INTERFACE I_DigitalInput EXTENDS I_Channel

PROPERTY P_Value : bool
GET
END_GET
END_PROPERTY

END_INTERFACE

(* stored: Version 1.1.0.1
   Itf I_DigitalInput: Id {214ef76f-f611-0f72-14f6-2b8f024fb231}
   Property P_Value: Id {ab716f7c-5ca4-0096-2327-73e953583b66}
   Get Get: Id {61283b4f-b50e-0dce-30ad-847da97974fa} *)
